# EPICS substitutions: bcmApp/Db/coefficientScaling.substitutions
file coefScale.db
{
pattern {P, AMC, COEF}

    {$(P), $(AMC), 0}
    {$(P), $(AMC), 1}

}
